# EPICS autosave request: ADProsilica/iocs/prosilicaIOC/iocBoot/iocProsilica/auto_settings.req
file "ADBase_settings.req",         P=$(P),  R=cam1:
file "prosilica_settings.req",      P=$(P),  R=cam1:
file "NDPluginBase_settings.req",   P=$(P),  R=image1:
file "NDStdArrays_settings.req",    P=$(P),  R=image1:
file "commonPlugin_settings.req",   P=$(P)
